INTERFACE I_MotionDrive

PROPERTY SaveAxisParams : BOOL
SET
END_SET
END_PROPERTY

END_INTERFACE

(* stored: Version 1.1.0.1
   Itf I_MotionDrive: Id {848572bc-fef8-4708-bb80-0dc37710e2cf}
   Property SaveAxisParams: Id {88e527c2-7636-499c-8190-d269c27617f6}
   Set Set: Id {7e245f11-24dd-4e06-ae0c-8fcdf753ea2b} *)
